TYPE ABSTRACT AxisBase_t :
STRUCT
    rActPos : REAL; // Current position
    bInPos  : SINT; // Current position index, 99=unknown
END_STRUCT
END_TYPE

(* stored: Version 1.1.0.1, ProductVersion 3.1.4024.6
   DUT AxisBase_t: Id {bcc92f59-cb67-4638-a1e0-6e3bbfb57cb3} *)
